// TIA Portal V19 export
VAR_GLOBAL   // PLC tag table "Em2"
END_VAR
VAR_GLOBAL CONSTANT   // user constants
   EM2_NO_OF_AXES : USInt := 2;   // Starts with 1. E.g., the value 4 means that 4 axes exist.
END_VAR
